TYPE stTarget :
STRUCT
	frame_id : eRefFrame;
	pose: ST_Pose;
END_STRUCT
END_TYPE

(* stored: Version 1.1.0.1, ProductVersion 3.1.4026.18
   DUT stTarget: Id {c1b2c3d4-2222-2222-2222-222222222222} *)
